Staubli VAL3: getName.pgx

public program getName(string& x_sName[], num x_nIndex)
begin
  x_sName=saveTool:name[x_nIndex]
end
